INTERFACE I_ReadParameter EXTENDS I_Status

PROPERTY AxisReadParamsInit : BOOL
GET
END_GET
END_PROPERTY

METHOD ReadParameters
VAR_INPUT
    Enable: BOOL;
    RefreshDelay: TIME;
END_VAR
END_METHOD

END_INTERFACE

(* stored: Version 1.1.0.1
   Itf I_ReadParameter: Id {44b7d62d-9b36-41c3-9b2a-5fe27104ee8d}
   Property AxisReadParamsInit: Id {aaa89008-d0c1-493e-a86d-8f92a0dabc9b}
   Get Get: Id {8bc2774e-5f18-4079-9b29-1c98c56a8fbb}
   Method ReadParameters: Id {9a4f678a-44d6-4f64-a6d1-07e4cd2a9e79} *)
